Omron CX-Programmer project NewProject (CX-Programmer 9.75)

# PLC Tangki: CJ2M CPU11

## Global symbols (name address type ; comment)
0.00 BOOL  ; UP
0.01 BOOL  ; DOWN
0.02 BOOL  ; RESET
100.00 BOOL  ; OUTPUT 1
100.01 BOOL  ; Q
C1 CHANNEL  ; COUNTER  1

## Program NewProgram1 (cyclic task 0)

### Section Section1

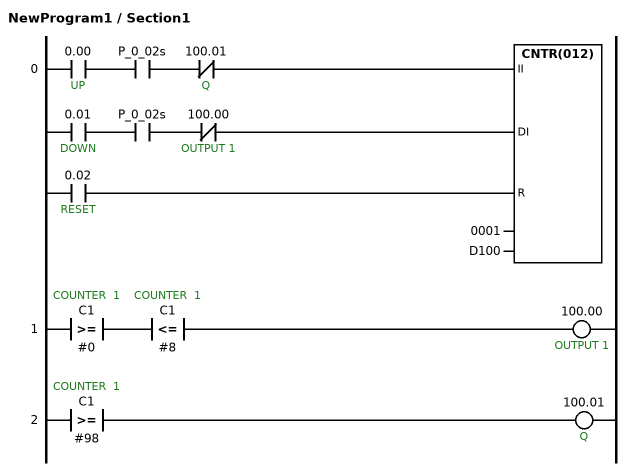
; rung 0
LD 0.00  ; UP
AND P_0_02s
ANDNOT 100.01  ; Q
LD 0.01  ; DOWN
AND P_0_02s
ANDNOT 100.00  ; OUTPUT 1
LD 0.02  ; RESET
CNTR(012) 0001 D100
; rung 1
LD>=(325) C1 #0  ; COUNTER  1
AND<=(315) C1 #8  ; COUNTER  1
OUT 100.00  ; OUTPUT 1
; rung 2
LD>=(325) C1 #98  ; COUNTER  1
OUT 100.01  ; Q
; rung 3
END(001)

### Section END
; rung 0
END(001)